% RSLogix 500 project P5 - Digital Rotameter.RSS, saved by version 8.30.00.16 %
PROJECT "P5"    % processor: Bul.1763 MicroLogix 1100 Series B %

PROGRAM FILES
  LAD 2 "MAIN"  8 rungs

DATA FILES
  O0 OUTPUT  4 elements
  I1 INPUT  6 elements
  S2 STATUS  66 elements
  B3 BINARY  1 elements
  T4 TIMER  1 elements
  C5 COUNTER  1 elements
  R6 CONTROL  1 elements
  N7 INTEGER  1 elements
  F8 FLOAT  3 elements

LADDER 2 "MAIN"
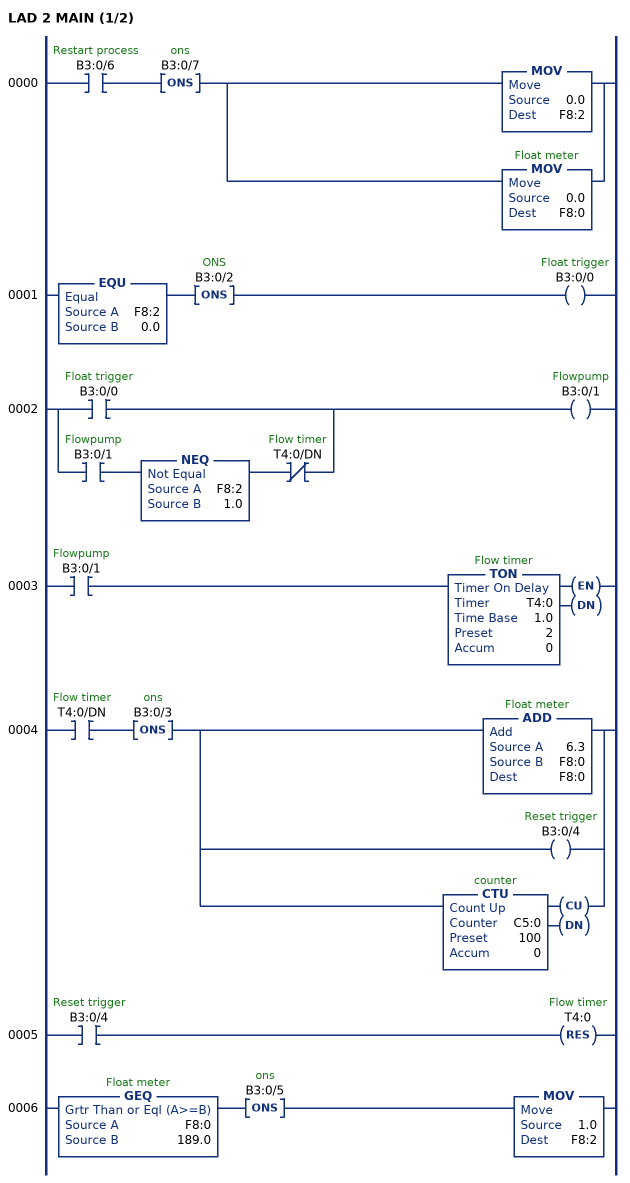
% Rung: 0 %
SOR XIC B3:0/6 ONS B3:0/7 BST MOV 0.0 F8:2 NXB MOV 0.0 F8:0 BND EOR
%   B3:0/6  "Restart process" %
%   B3:0/7  "ons" %
%   F8:0  "Float meter" %
% Rung: 1 %
SOR EQU F8:2 0.0 ONS B3:0/2 OTE B3:0/0 EOR
%   B3:0/2  "ONS" %
%   B3:0/0  "Float trigger" %
% Rung: 2 %
SOR BST XIC B3:0/0 NXB XIC B3:0/1 NEQ F8:2 1.0 XIO T4:0/DN BND OTE B3:0/1 EOR
%   B3:0/0  "Float trigger" %
%   B3:0/1  "Flowpump" %
%   T4:0  "Flow timer" %
% Rung: 3 %
SOR XIC B3:0/1 TON T4:0 1.0 2 0 EOR
%   B3:0/1  "Flowpump" %
%   T4:0  "Flow timer" %
% Rung: 4 %
SOR XIC T4:0/DN ONS B3:0/3 BST ADD 6.3 F8:0 F8:0 NXB OTE B3:0/4 NXB CTU C5:0 100 0 BND EOR
%   T4:0  "Flow timer" %
%   B3:0/3  "ons" %
%   F8:0  "Float meter" %
%   B3:0/4  "Reset trigger" %
%   C5:0  "counter" %
% Rung: 5 %
SOR XIC B3:0/4 RES T4:0 EOR
%   B3:0/4  "Reset trigger" %
%   T4:0  "Flow timer" %
% Rung: 6 %
SOR GEQ F8:0 189.0 ONS B3:0/5 MOV 1.0 F8:2 EOR
%   F8:0  "Float meter" %
%   B3:0/5  "ons" %

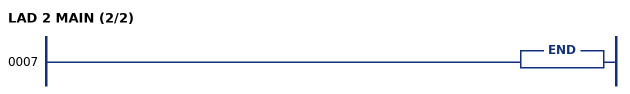
% Rung: 7 %
SOR END EOR

OTHER DOCUMENTED ADDRESSES
  F8:1  "Holder"

DATA TABLE (non-zero values as saved)
DATA T4
% .PRE .ACC %
% T4:0 % 2 0
DATA C5
% .PRE .ACC %
% C5:0 % 100 0
